(* PLC project Cell Example , CTH FIX1 1.0, author CTH SS2 *)
(* stored: companyURL www.chalmers.se, creationDateTime 2008-03-19T20:31:26, version 1.0, modificationDateTime 2008-05-30T23:21:46, organization SS2, language en-US *)

TYPE BinaryPositions : ();
END_TYPE

FUNCTION ADD_E : INT
  VAR_INPUT
    Enable : BOOL := FALSE;
    IN1 : INT := 0;
    IN2 : INT := 0;
  END_VAR
  VAR_OUTPUT
    EnableO : BOOL := FALSE;
  END_VAR

(* LD diagram, written out as Structured Text *)
END_FUNCTION

FUNCTION DEC_E : INT
  VAR_INPUT
    Enable : BOOL;
  END_VAR
  VAR_OUTPUT
    EnableO : BOOL;
  END_VAR

(* LD diagram, written out as Structured Text *)
END_FUNCTION

FUNCTION MOVE_E : STRING
  VAR_INPUT
    Enable : BOOL := FALSE;
    IN : STRING;
  END_VAR
  VAR_OUTPUT
    EnableO : BOOL := FALSE;
  END_VAR

(* LD diagram, written out as Structured Text *)
END_FUNCTION

FUNCTION_BLOCK test4
  VAR_INPUT
    i1 : BOOL := FALSE;
  END_VAR
  VAR_OUTPUT
    o1 : BOOL := TRUE;
  END_VAR

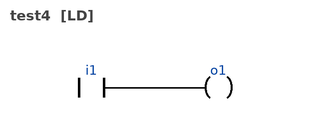
(* LD diagram, written out as Structured Text *)
o1 := i1;
END_FUNCTION_BLOCK

FUNCTION_BLOCK test2
  VAR_INPUT
    i : BOOL;
  END_VAR
  VAR_OUTPUT
    o : BOOL;
  END_VAR
  VAR
    internal1 : test4;
  END_VAR

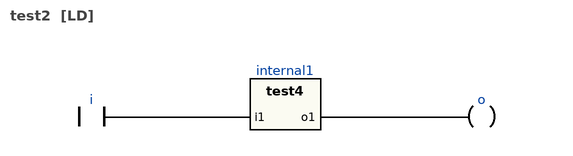
(* LD diagram, written out as Structured Text *)
internal1(i1 := i);
o := internal1.o1;
END_FUNCTION_BLOCK

FUNCTION_BLOCK test5
  VAR_INPUT
    in : BOOL;
  END_VAR
  VAR_OUTPUT
    ut : BOOL;
  END_VAR

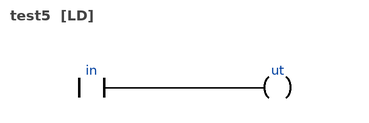
(* LD diagram, written out as Structured Text *)
ut := in;
END_FUNCTION_BLOCK

FUNCTION_BLOCK test3
  VAR_INPUT
    in1 : BOOL;
  END_VAR
  VAR_OUTPUT
    ut1 : BOOL;
  END_VAR
  VAR
    internal1 : test4;
    internal2 : test5;
  END_VAR

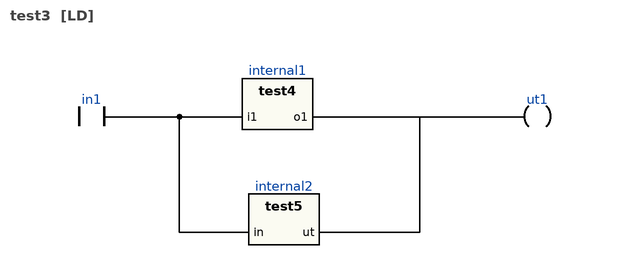
(* LD diagram, written out as Structured Text *)
internal1(i1 := in1);
internal2(in := in1);
ut1 := internal1.o1 OR internal2.ut;
END_FUNCTION_BLOCK

FUNCTION_BLOCK TestFB
  VAR_INPUT
    IN1 : BOOL := FALSE;
    IN2 : INT := 0;
    IN3 : BOOL := FALSE;
  END_VAR
  VAR_OUTPUT
    OUT1 : BOOL := FALSE;
    OUT2 : BOOL := FALSE;
    OUT3 : BOOL := FALSE;
    OUT4 : INT := 0;
  END_VAR
  VAR
    internal1 : test2;
    internal2 : test3;
  END_VAR

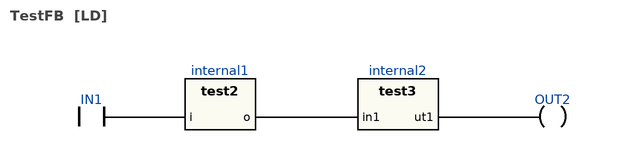
(* LD diagram, written out as Structured Text *)
internal1(i := IN1);
internal2(in1 := internal1.o);
OUT2 := internal2.ut1;
END_FUNCTION_BLOCK

FUNCTION_BLOCK RAC
  VAR_INPUT
    IN1 : BOOL := FALSE;
  END_VAR
  VAR_OUTPUT
    OUT : BOOL := FALSE;
  END_VAR
  VAR_INPUT
    IN2 : BOOL := TRUE;
  END_VAR
  VAR
    Var3 : BOOL := TRUE;
    IN4 : INT := 5;
  END_VAR
  VAR_OUTPUT
    State : STRING := 'Undefined';
  END_VAR
  VAR
    timer : TON;
    passedTime : TIME := 20;
    test : TestFB;
  END_VAR
  VAR_OUTPUT
    OUT2 : BOOL := TRUE;
  END_VAR
  VAR  (* added by the conversion: wires and edge detectors of the diagram *)
    _ADD_E24_ : ANY;
    _ADD_E24_OUT : INT;
    _MOVE_E26_ : ANY;
    _MOVE_E26_OUT : STRING;
    _DEC_E34_ : ANY;
    _DEC_E34_OUT : INT;
  END_VAR

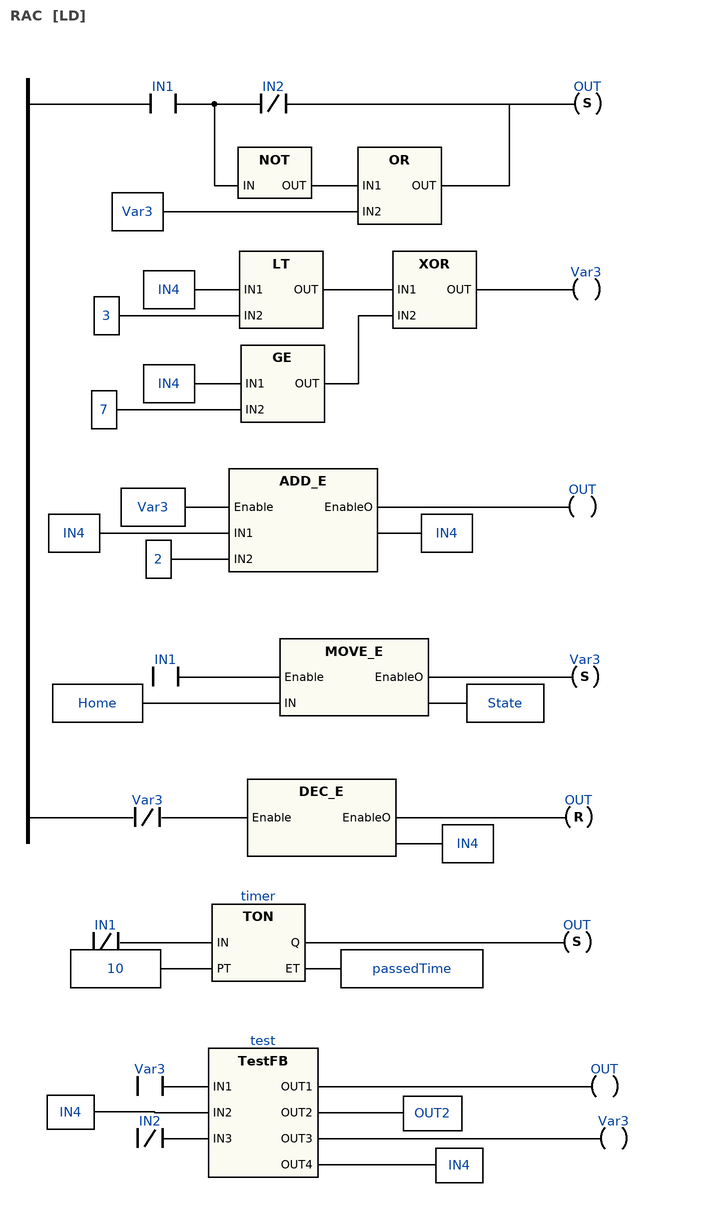
(* LD diagram, written out as Structured Text *)
IF IN1 AND NOT IN2 OR NOT IN1 OR Var3 THEN OUT := TRUE; END_IF;
Var3 := IN4 < 3 XOR IN4 >= 7;
_ADD_E24_OUT := ADD_E(Enable := Var3, IN1 := IN4, IN2 := 2,  => _ADD_E24_);
OUT := _ADD_E24_OUT;
IN4 := _ADD_E24_OUT;
_MOVE_E26_OUT := MOVE_E(Enable := IN1, IN := Home,  => _MOVE_E26_);
IF _MOVE_E26_OUT THEN Var3 := TRUE; END_IF;
State := _MOVE_E26_OUT;
_DEC_E34_OUT := DEC_E(Enable := NOT Var3,  => _DEC_E34_);
IF _DEC_E34_OUT THEN OUT := FALSE; END_IF;
IN4 := _DEC_E34_OUT;
timer(IN := NOT IN1, PT := 10);
IF timer.Q THEN OUT := TRUE; END_IF;
passedTime := timer.ET;
test(IN1 := Var3, IN2 := IN4, IN3 := NOT IN2);
OUT := test.OUT1;
OUT2 := test.OUT2;
Var3 := test.OUT3;
IN4 := test.OUT4;
END_FUNCTION_BLOCK

FUNCTION INCP_M : INT
  VAR_INPUT
    Enable : BOOL := FALSE;
  END_VAR
  VAR_OUTPUT
    EnableO : BOOL := FALSE;
  END_VAR

(* LD diagram, written out as Structured Text *)
END_FUNCTION

FUNCTION MOV_M : INT
  VAR_INPUT
    Enable : BOOL := FALSE;
    s_in : INT := 0;
  END_VAR
  VAR_OUTPUT
    EnableO : BOOL := FALSE;
  END_VAR

(* LD diagram, written out as Structured Text *)
END_FUNCTION

FUNCTION_BLOCK FB_Event
  VAR_INPUT
    Dig_in : BOOL := FALSE;
  END_VAR
  VAR_OUTPUT
    Dig_Ut : BOOL := FALSE;
  END_VAR
  VAR
    Tid_Klar : BOOL := 0;
    Tmp_INT : INT := FALSE;
    Dig_Ut_c : BOOL := FALSE;
    Counting : BOOL := FALSE;
  END_VAR
  VAR  (* added by the conversion: wires and edge detectors of the diagram *)
    _MOV_M7_ : ANY;
    _MOV_M7_OUT : INT;
    _INCP_M13_ : ANY;
    _INCP_M13_OUT : INT;
  END_VAR

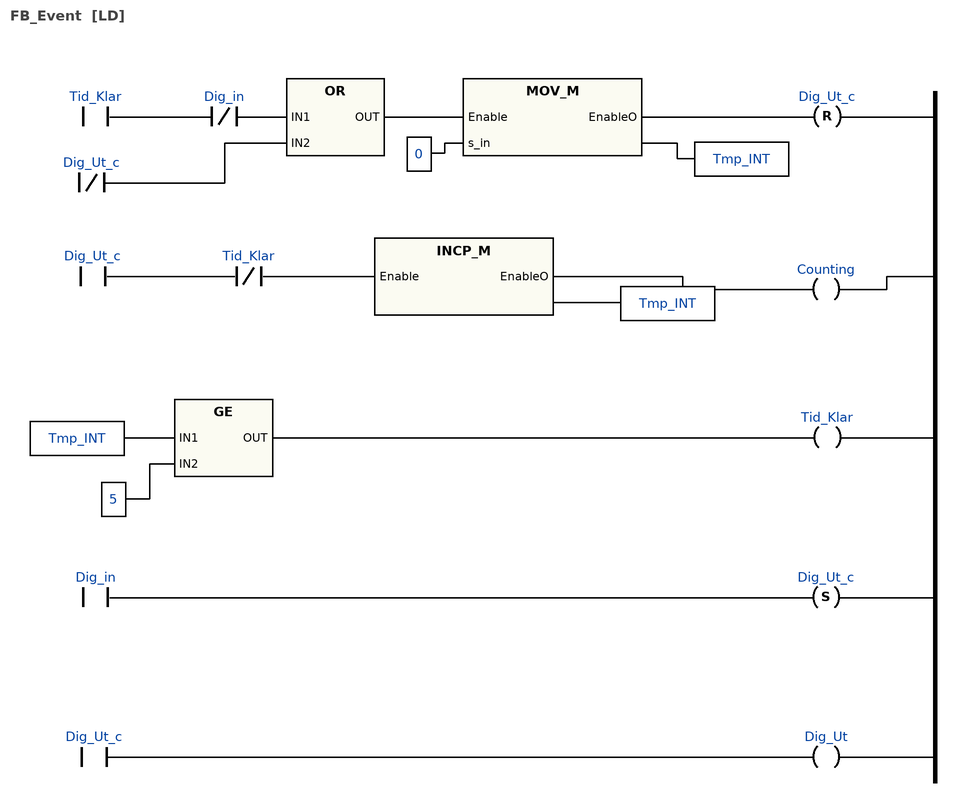
(* LD diagram, written out as Structured Text *)
_MOV_M7_OUT := MOV_M(Enable := Tid_Klar AND NOT Dig_in OR NOT Dig_Ut_c, s_in := 0,  => _MOV_M7_);
IF _MOV_M7_OUT THEN Dig_Ut_c := FALSE; END_IF;
Tmp_INT := _MOV_M7_OUT;
_INCP_M13_OUT := INCP_M(Enable := Dig_Ut_c AND NOT Tid_Klar,  => _INCP_M13_);
Tmp_INT := _INCP_M13_OUT;
Counting := _INCP_M13_OUT;
Tid_Klar := Tmp_INT >= 5;
IF Dig_in THEN Dig_Ut_c := TRUE; END_IF;
Dig_Ut := Dig_Ut_c;
END_FUNCTION_BLOCK

FUNCTION_BLOCK TIMER_100_FB_M
  VAR_INPUT
    Coil : BOOL := FALSE;
    Preset : INT := 0;
    ValueIn : INT := 0;
  END_VAR
  VAR_OUTPUT
    ValueOut : INT := 0;
    Status : BOOL := FALSE;
  END_VAR

(* LD diagram, written out as Structured Text *)
END_FUNCTION_BLOCK

FUNCTION_BLOCK FB_Move_533
  VAR_INPUT
    Enable : BOOL := FALSE;
    Hand : BOOL := FALSE;
    HandFwd : BOOL := FALSE;
    HandRev : BOOL := FALSE;
    Auto : BOOL := FALSE;
    AutoFwd : BOOL := FALSE;
    AutoRev : BOOL := FALSE;
    EndPosFwd : BOOL := FALSE;
    EndPosRev : BOOL := FALSE;
    InterlockFwd : BOOL := FALSE;
    InterlockRev : BOOL := FALSE;
    SetRst : BOOL := FALSE;
    TimeValue : INT := 10;
  END_VAR
  VAR
    McOutputFwd : BOOL := FALSE;
    McOutputRev : BOOL := FALSE;
    McFwd : BOOL := FALSE;
    McRev : BOOL := FALSE;
    OutputFwd : BOOL := FALSE;
    OutputRev : BOOL := FALSE;
    TimeOutFwd : BOOL := FALSE;
  END_VAR
  VAR_OUTPUT
    TimeOutRev : BOOL := FALSE;
    EventFwd : BOOL := FALSE;
    EventRev : BOOL := FALSE;
  END_VAR
  VAR
    Event_Rev : FB_Event;
    Event_Fwd : FB_Event;
    TimerRev : TIMER_100_FB_M;
    TimerFwd : TIMER_100_FB_M;
  END_VAR

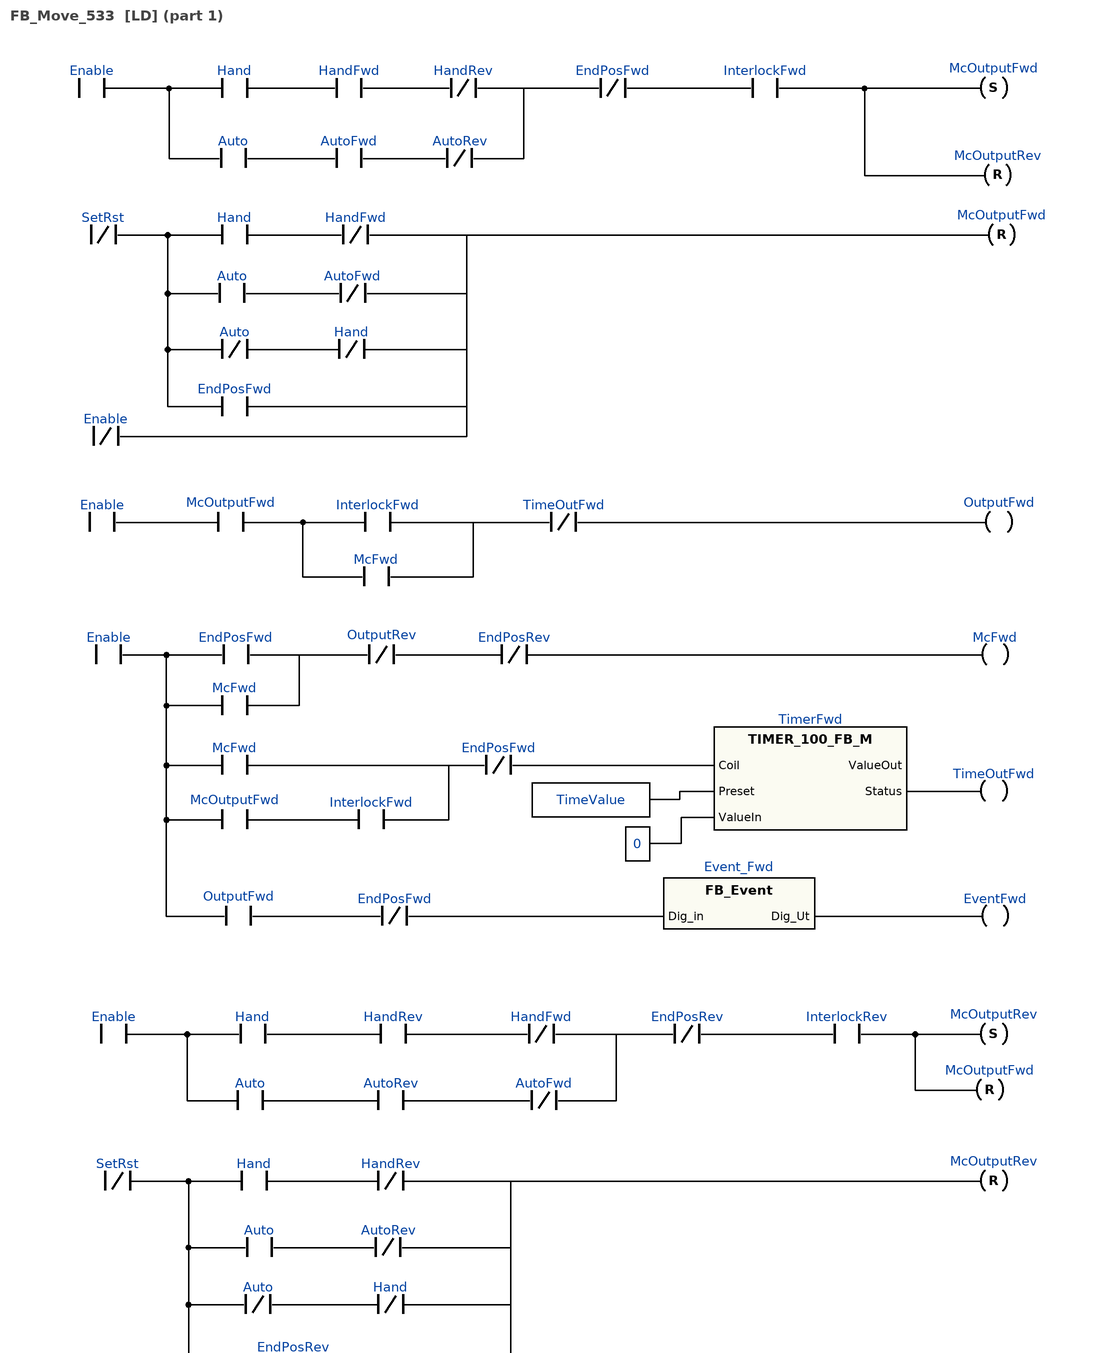
(* LD diagram, written out as Structured Text *)
IF Enable AND (Auto AND AutoFwd AND NOT AutoRev OR Hand AND HandFwd AND NOT HandRev) AND NOT EndPosFwd AND InterlockFwd THEN McOutputFwd := TRUE; END_IF;
IF Enable AND (Auto AND AutoFwd AND NOT AutoRev OR Hand AND HandFwd AND NOT HandRev) AND NOT EndPosFwd AND InterlockFwd THEN McOutputRev := FALSE; END_IF;
IF NOT SetRst AND Hand AND NOT HandFwd OR NOT SetRst AND Auto AND NOT AutoFwd OR NOT SetRst AND NOT Auto AND NOT Hand OR NOT SetRst AND EndPosFwd OR NOT Enable THEN McOutputFwd := FALSE; END_IF;
OutputFwd := Enable AND McOutputFwd AND (InterlockFwd OR McFwd) AND NOT TimeOutFwd;
McFwd := Enable AND (McFwd OR EndPosFwd) AND NOT OutputRev AND NOT EndPosRev;
TimerFwd(Coil := Enable AND (McFwd OR McOutputFwd AND InterlockFwd) AND NOT EndPosFwd, Preset := TimeValue, ValueIn := 0);
TimeOutFwd := TimerFwd.Status;
Event_Fwd(Dig_in := Enable AND OutputFwd AND NOT EndPosFwd);
EventFwd := Event_Fwd.Dig_Ut;
IF Enable AND (Hand AND HandRev AND NOT HandFwd OR Auto AND AutoRev AND NOT AutoFwd) AND NOT EndPosRev AND InterlockRev THEN McOutputRev := TRUE; END_IF;
IF Enable AND (Hand AND HandRev AND NOT HandFwd OR Auto AND AutoRev AND NOT AutoFwd) AND NOT EndPosRev AND InterlockRev THEN McOutputFwd := FALSE; END_IF;
IF NOT SetRst AND Hand AND NOT HandRev OR NOT SetRst AND Auto AND NOT AutoRev OR NOT SetRst AND NOT Auto AND NOT Hand OR NOT SetRst AND EndPosRev OR NOT Enable THEN McOutputRev := FALSE; END_IF;
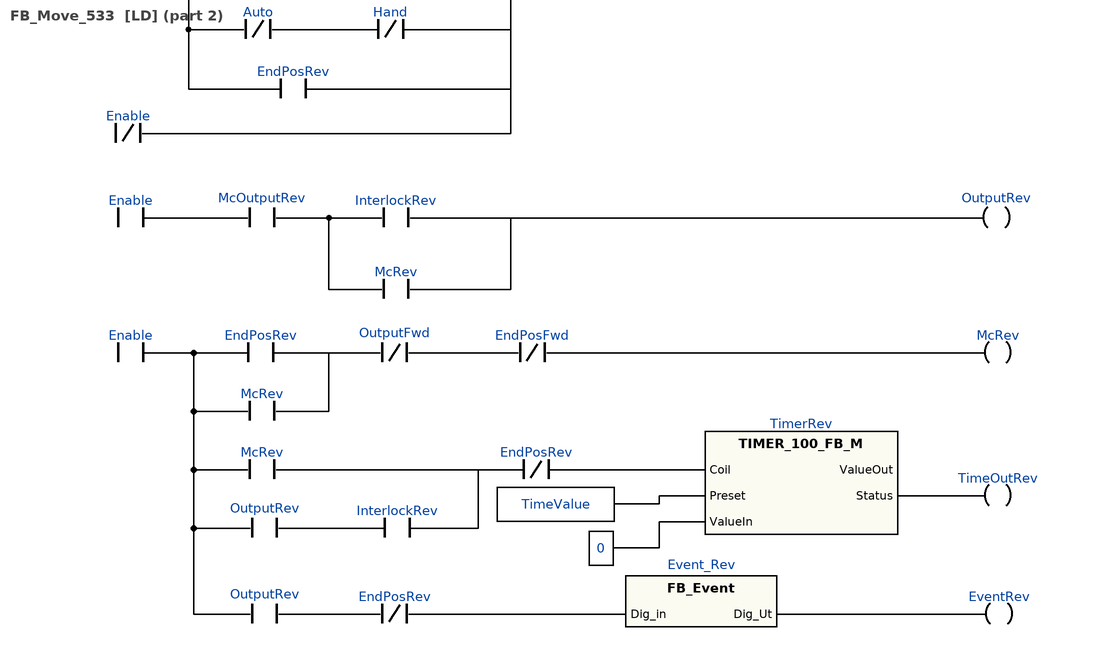
OutputRev := Enable AND McOutputRev AND (InterlockRev OR McRev);
McRev := Enable AND (EndPosRev OR McRev) AND NOT OutputFwd AND NOT EndPosFwd;
TimerRev(Coil := Enable AND (McRev OR OutputRev AND InterlockRev) AND NOT EndPosRev, Preset := TimeValue, ValueIn := 0);
TimeOutRev := TimerRev.Status;
Event_Rev(Dig_in := Enable AND OutputRev AND NOT EndPosRev);
EventRev := Event_Rev.Dig_Ut;
END_FUNCTION_BLOCK

CONFIGURATION ExampleCell
END_CONFIGURATION
